// TIA Portal project "Szablon_Finał_V17" (V17)

(* hardware
DEVICE "S7-1200 station_1"  S7-1200 Station
   slot 0: "Rack_0"  S7-1200 Rack  Rack  V1.0
   slot 1: "PLC_1"  CPU 1214C DC/DC/DC  6ES7 214-1AG40-0XB0  V4.2
*)

// ===== PLC "PLC_1"  CPU 1214C DC/DC/DC =====

VAR_GLOBAL   // PLC tag table "Default tag table"
   "minimum" AT %I0.0 : Bool;
   "maksimum" AT %I0.1 : Bool;
   "poziom A" AT %I0.2 : Bool;
   "minimum B" AT %I0.3 : Bool;
   "Pokrywa" AT %I0.4 : Bool;
   "Start" AT %I0.5 : Bool;
   "Stop awaryjny" AT %I0.6 : Bool;
   "Zwolnij alarm" AT %I0.7 : Bool;
   "Mieszadło M1" AT %Q0.0 : Bool;
   "Mieszadło M2" AT %Q0.1 : Bool;
   "Zawór Z1" AT %Q0.2 : Bool;
   "Zawór Z2" AT %Q0.3 : Bool;
   "Zawór Z3" AT %Q0.4 : Bool;
   "Pompa P" AT %Q0.5 : Bool;
   "Alarm" AT %Q0.6 : Bool;
   "Tag_1" AT %MW50 : Int;
END_VAR

DATA_BLOCK "Dwa zbiorniki_DB"   // DB6
{ S7_Optimized_Access := 'TRUE' }
VERSION : 0.1
// stored: InstanceOfName Dwa zbiorniki
"Dwa zbiorniki"
BEGIN
END_DATA_BLOCK

DATA_BLOCK "Mieszanie substancji_DB"   // DB10
{ S7_Optimized_Access := 'TRUE' }
VERSION : 0.1
// stored: InstanceOfName Mieszanie substancji
"Mieszanie substancji"
BEGIN
END_DATA_BLOCK

// folder: System blocks/Program resources

DATA_BLOCK "IEC_Timer_0_DB"   // DB1
{ S7_Optimized_Access := 'TRUE' }
AUTHOR : Simatic
FAMILY : IEC
NAME : IEC_TMR
VERSION : 1.0
// stored: InstanceOfName IEC_TIMER
"IEC_TIMER"
BEGIN
END_DATA_BLOCK

DATA_BLOCK "IEC_Timer_0_DB_1"   // DB2
{ S7_Optimized_Access := 'TRUE' }
AUTHOR : Simatic
FAMILY : IEC
NAME : IEC_TMR
VERSION : 1.0
// stored: InstanceOfName IEC_TIMER
"IEC_TIMER"
BEGIN
END_DATA_BLOCK

DATA_BLOCK "IEC_Timer_0_DB_2"   // DB3
{ S7_Optimized_Access := 'TRUE' }
AUTHOR : Simatic
FAMILY : IEC
NAME : IEC_TMR
VERSION : 1.0
// stored: InstanceOfName IEC_TIMER
"IEC_TIMER"
BEGIN
END_DATA_BLOCK

DATA_BLOCK "IEC_Timer_0_DB_3"   // DB4
{ S7_Optimized_Access := 'TRUE' }
AUTHOR : Simatic
FAMILY : IEC
NAME : IEC_TMR
VERSION : 1.0
// stored: InstanceOfName IEC_TIMER
"IEC_TIMER"
BEGIN
END_DATA_BLOCK

DATA_BLOCK "IEC_Timer_0_DB_4"   // DB5
{ S7_Optimized_Access := 'TRUE' }
AUTHOR : Simatic
FAMILY : IEC
NAME : IEC_TMR
VERSION : 1.0
// stored: InstanceOfName IEC_TIMER
"IEC_TIMER"
BEGIN
END_DATA_BLOCK

DATA_BLOCK "IEC_Timer_0_DB_5"   // DB7
{ S7_Optimized_Access := 'TRUE' }
AUTHOR : Simatic
FAMILY : IEC
NAME : IEC_TMR
VERSION : 1.0
// stored: InstanceOfName IEC_TIMER
"IEC_TIMER"
BEGIN
END_DATA_BLOCK

DATA_BLOCK "IEC_Timer_0_DB_6"   // DB8
{ S7_Optimized_Access := 'TRUE' }
AUTHOR : Simatic
FAMILY : IEC
NAME : IEC_TMR
VERSION : 1.0
// stored: InstanceOfName IEC_TIMER
"IEC_TIMER"
BEGIN
END_DATA_BLOCK

DATA_BLOCK "IEC_Timer_0_DB_7"   // DB9
{ S7_Optimized_Access := 'TRUE' }
AUTHOR : Simatic
FAMILY : IEC
NAME : IEC_TMR
VERSION : 1.0
// stored: InstanceOfName IEC_TIMER
"IEC_TIMER"
BEGIN
END_DATA_BLOCK

// folder: (top level)

FUNCTION_BLOCK "Dwa zbiorniki"   // FB1, LAD
{ S7_Optimized_Access := 'TRUE' }
VERSION : 0.1
   VAR_INPUT
      minimum : Bool;
      maximum : Bool;
      "poziom A" : Bool;
      "minimum B" : Bool;
      Pokrywa : Bool;
      Start : Bool;
      "Stop awaryjny" : Bool;
      "Zwolnij alarm" : Bool;
   END_VAR
   VAR_OUTPUT
      M1 : Bool;
      M2 : Bool;
      "Pompa P" : Bool;
      Alarm : Bool;
   END_VAR
   VAR_IN_OUT
      Z1 : Bool;
      Z2 : Bool;
      Z3 : Bool;
      State : Int;
   END_VAR
   VAR
      Start_edge : Bool;
      Stop_awaryjny_edge : Bool;
      Zwolnij_alarm_edge : Bool;
   END_VAR
   VAR_TEMP
      "alarm 0_5Hz" : Bool;
      "alarm 1Hz" : Bool;
      alarm_awaryjny : Bool;
   END_VAR
   VAR_TEMP   // added for the SCL form of the ladder/FBD networks
      _w1 : Bool;
      _w2 : Bool;
   END_VAR
BEGIN

REGION Network 1
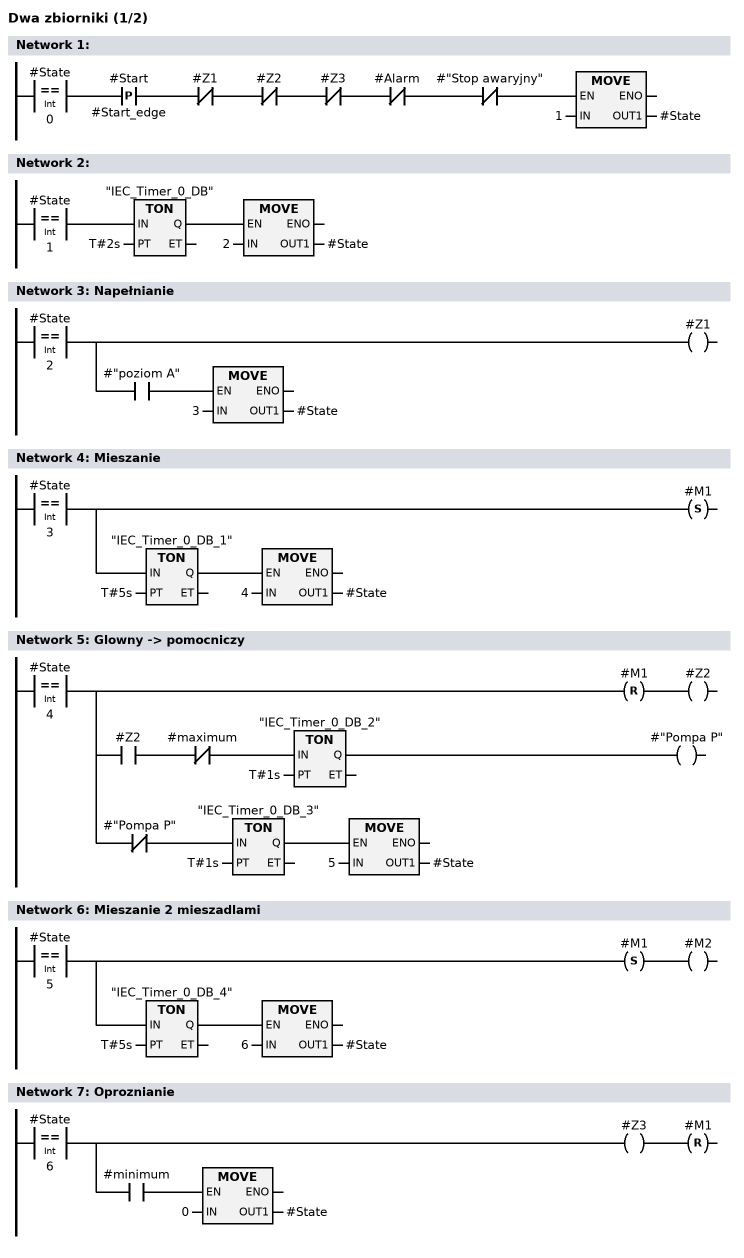
   RUNG wire#powerrail
      { S7_Templates := "SrcType := Int" } EQ_Contact(in1 := #State, in2 := 0)
      P_Contact(operand := #Start, bit := #Start_edge)
      I_Contact( #Z1 )
      I_Contact( #Z2 )
      I_Contact( #Z3 )
      I_Contact( #Alarm )
      I_Contact( #"Stop awaryjny" )
      Move(in := 1, out1 => #State)
   END_RUNG
   // the same network as SCL:
   #_w1 := (#State = 0) AND #Start AND NOT #Start_edge;   // rising edge of #Start
   #Start_edge := #Start;
   IF #_w1 AND NOT #Z1 AND NOT #Z2 AND NOT #Z3 AND NOT #Alarm AND NOT #"Stop awaryjny" THEN
       #State := 1;
   END_IF;
END_REGION

REGION Network 2
   "IEC_Timer_0_DB".TON(IN := #State = 1, PT := T#2s);
   IF "IEC_Timer_0_DB".Q THEN #State := 2; END_IF;
END_REGION

REGION Network 3: Napełnianie
   RUNG wire#powerrail
      { S7_Templates := "SrcType := Int" } EQ_Contact(in1 := #State, in2 := 2)
      wire#w1
      Coil( #Z1 )
   END_RUNG
   RUNG wire#w1
      Contact( #"poziom A" )
      Move(in := 3, out1 => #State)
   END_RUNG
   // the same network as SCL:
   #Z1 := #State = 2;
   IF #Z1 AND #"poziom A" THEN #State := 3; END_IF;
END_REGION

REGION Network 4: Mieszanie
   #_w1 := #State = 3;
   IF #_w1 THEN #M1 := TRUE; END_IF;
   "IEC_Timer_0_DB_1".TON(IN := #_w1, PT := T#5s);
   IF "IEC_Timer_0_DB_1".Q THEN #State := 4; END_IF;
END_REGION

REGION Network 5: Glowny -> pomocniczy
   #_w1 := #State = 4;
   IF #_w1 THEN #M1 := FALSE; END_IF;
   #Z2 := #_w1;
   "IEC_Timer_0_DB_2".TON(IN := #_w1 AND #Z2 AND NOT #maximum, PT := T#1s);
   #"Pompa P" := "IEC_Timer_0_DB_2".Q;
   "IEC_Timer_0_DB_3".TON(IN := #_w1 AND NOT #"Pompa P", PT := T#1s);
   IF "IEC_Timer_0_DB_3".Q THEN #State := 5; END_IF;
END_REGION

REGION Network 6: Mieszanie 2 mieszadlami
   #_w1 := #State = 5;
   IF #_w1 THEN #M1 := TRUE; END_IF;
   #M2 := #_w1;
   "IEC_Timer_0_DB_4".TON(IN := #_w1, PT := T#5s);
   IF "IEC_Timer_0_DB_4".Q THEN #State := 6; END_IF;
END_REGION

REGION Network 7: Oproznianie
   RUNG wire#powerrail
      { S7_Templates := "SrcType := Int" } EQ_Contact(in1 := #State, in2 := 6)
      wire#w1
      Coil( #Z3 )
      R_Coil( #M1 )
   END_RUNG
   RUNG wire#w1
      Contact( #minimum )
      Move(in := 0, out1 => #State)
   END_RUNG
   // the same network as SCL:
   #Z3 := #State = 6;
   IF #Z3 THEN #M1 := FALSE; END_IF;
   IF #Z3 AND #minimum THEN #State := 0; END_IF;
END_REGION

REGION Network 8: f = 0.5Hz, duty = 25%
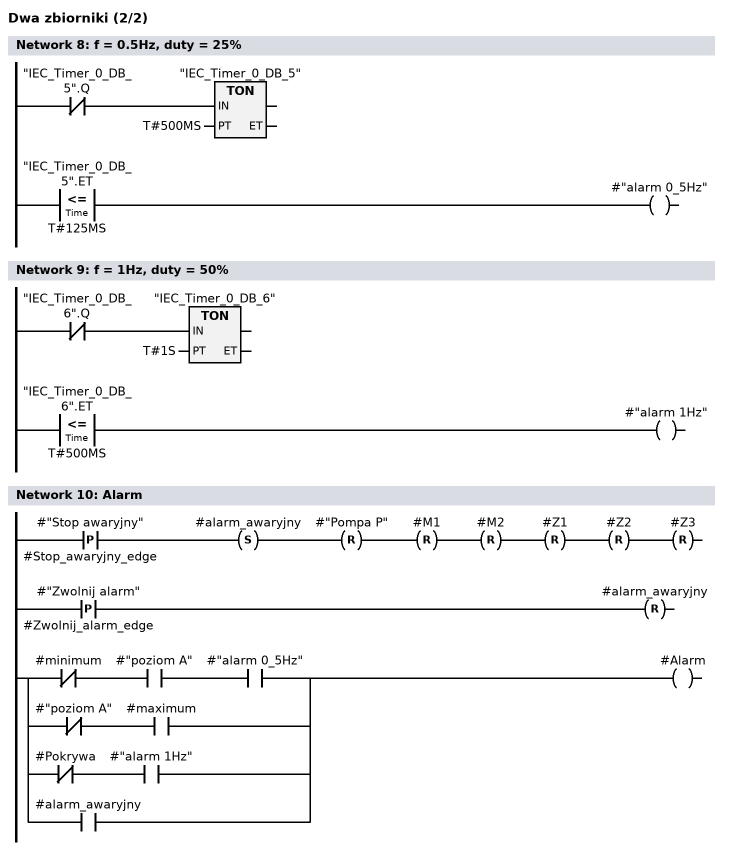
   "IEC_Timer_0_DB_5".TON(IN := NOT "IEC_Timer_0_DB_5".Q, PT := T#500MS);
   #"alarm 0_5Hz" := "IEC_Timer_0_DB_5".ET <= T#125MS;
END_REGION

REGION Network 9: f = 1Hz, duty = 50%
   "IEC_Timer_0_DB_6".TON(IN := NOT "IEC_Timer_0_DB_6".Q, PT := T#1S);
   #"alarm 1Hz" := "IEC_Timer_0_DB_6".ET <= T#500MS;
END_REGION

REGION Network 10: Alarm
   RUNG wire#powerrail
      P_Contact(operand := #"Stop awaryjny", bit := #Stop_awaryjny_edge)
      S_Coil( #alarm_awaryjny )
      R_Coil( #"Pompa P" )
      R_Coil( #M1 )
      R_Coil( #M2 )
      R_Coil( #Z1 )
      R_Coil( #Z2 )
      R_Coil( #Z3 )
   END_RUNG
   RUNG wire#powerrail
      P_Contact(operand := #"Zwolnij alarm", bit := #Zwolnij_alarm_edge)
      R_Coil( #alarm_awaryjny )
   END_RUNG
   RUNG wire#powerrail
      I_Contact( #minimum )
      Contact( #"poziom A" )
      Contact( #"alarm 0_5Hz" )
      wire#w1
      Coil( #Alarm )
   END_RUNG
   RUNG wire#powerrail
      I_Contact( #"poziom A" )
      Contact( #maximum )
   END_RUNG wire#w1
   RUNG wire#powerrail
      I_Contact( #Pokrywa )
      Contact( #"alarm 1Hz" )
   END_RUNG wire#w1
   RUNG wire#powerrail
      Contact( #alarm_awaryjny )
   END_RUNG wire#w1
   // the same network as SCL:
   #_w1 := #"Stop awaryjny" AND NOT #Stop_awaryjny_edge;   // rising edge of #"Stop awaryjny"
   #Stop_awaryjny_edge := #"Stop awaryjny";
   IF #_w1 THEN
       #alarm_awaryjny := TRUE;
       #"Pompa P" := FALSE;
       #M1 := FALSE;
       #M2 := FALSE;
       #Z1 := FALSE;
       #Z2 := FALSE;
       #Z3 := FALSE;
   END_IF;
   #_w2 := #"Zwolnij alarm" AND NOT #Zwolnij_alarm_edge;   // rising edge of #"Zwolnij alarm"
   #Zwolnij_alarm_edge := #"Zwolnij alarm";
   IF #_w2 THEN #alarm_awaryjny := FALSE; END_IF;
   #Alarm := (NOT #minimum AND #"poziom A" AND #"alarm 0_5Hz") OR (NOT #"poziom A" AND #maximum) OR (NOT #Pokrywa AND #"alarm 1Hz") OR #alarm_awaryjny;
END_REGION
END_FUNCTION_BLOCK

FUNCTION_BLOCK "Mieszanie substancji"   // FB2, LAD
{ S7_Optimized_Access := 'TRUE' }
VERSION : 0.1
   VAR_OUTPUT
      A_percent : Real;
      B_percent : Real;
      C_percent : Real;
      AF001 : Bool;
      AF002 : Bool;
      AF003 : Bool;
      AF004 : Bool;
      AF005 : Bool;
      AF006 : Bool;
      AF007 : Bool;
      AF008 : Bool;
   END_VAR
   VAR_IN_OUT
      A_value : Int := 2500;
      B_value : Int := 2500;
      C_value : Int := 9000;
      M_value : Int := 12;
   END_VAR
   VAR
      TON_Out : Bool;
      State : Int;
      TON_Out_edge : Bool;
      A_in_M : Int;
      B_in_M : Int;
      C_in_M : Int;
      TON_Out_edge2 : Bool;
   END_VAR
   VAR CONSTANT
      qa : Int := 4;
      qb : Int := 8;
      qc : Int := 12;
      qabc : Int := 15;
   END_VAR
   VAR_TEMP   // added for the SCL form of the ladder/FBD networks
      _w1 : Bool;
      _w2 : Bool;
   END_VAR
BEGIN

REGION Network 1
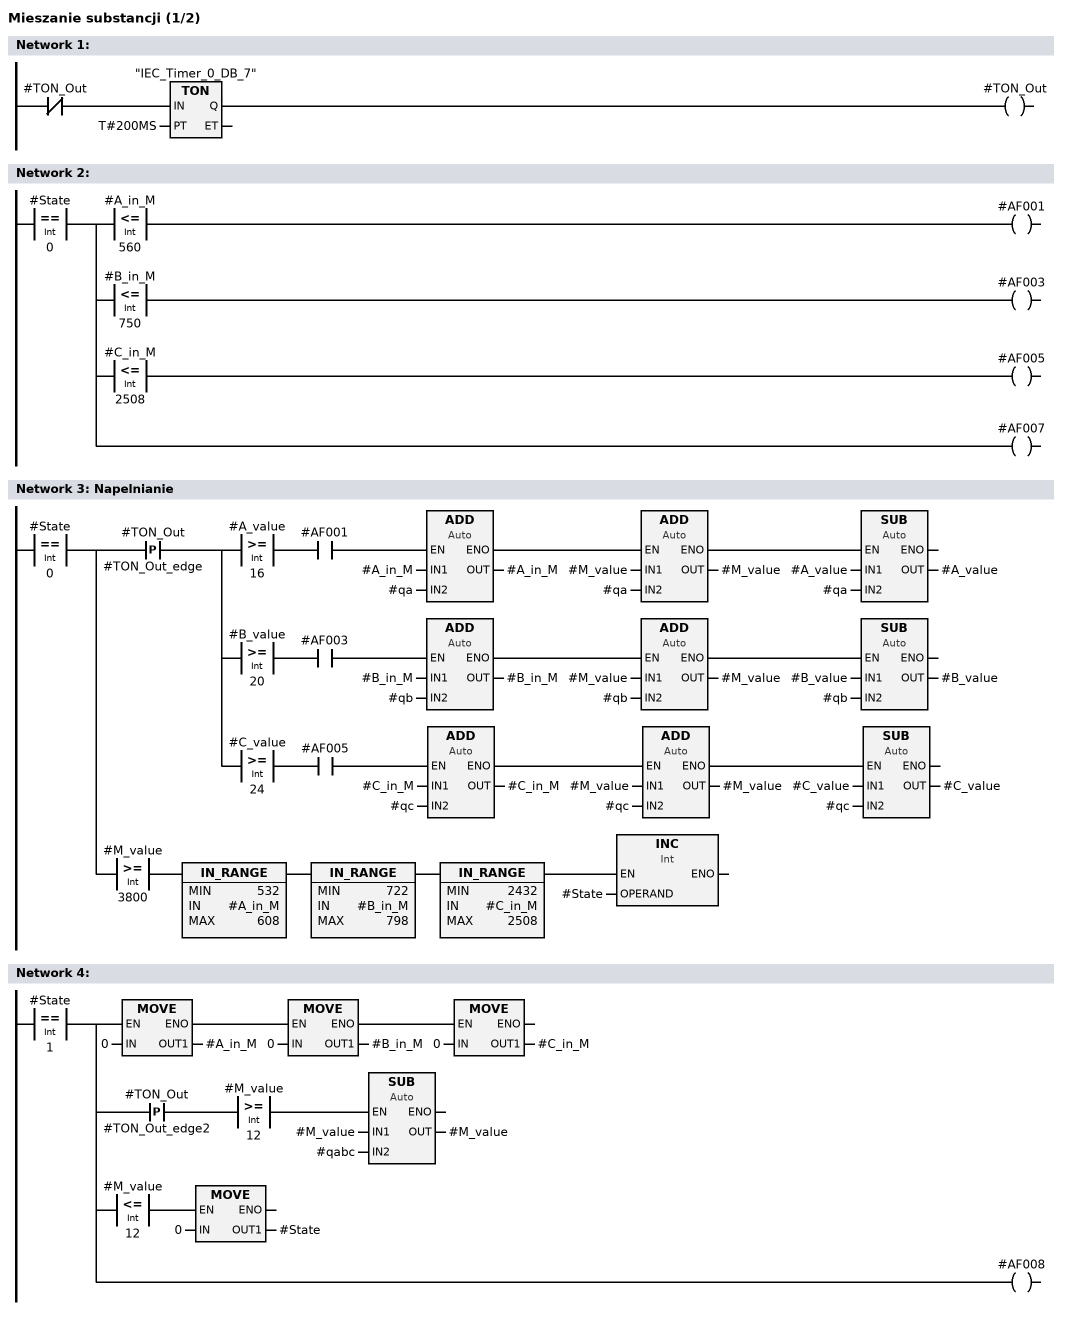
   "IEC_Timer_0_DB_7".TON(IN := NOT #TON_Out, PT := T#200MS);
   #TON_Out := "IEC_Timer_0_DB_7".Q;
END_REGION

REGION Network 2
   RUNG wire#powerrail
      { S7_Templates := "SrcType := Int" } EQ_Contact(in1 := #State, in2 := 0)
      wire#w1
      { S7_Templates := "SrcType := Int" } LE_Contact(in1 := #A_in_M, in2 := 560)
      Coil( #AF001 )
   END_RUNG
   RUNG wire#w1
      { S7_Templates := "SrcType := Int" } LE_Contact(in1 := #B_in_M, in2 := 750)
      Coil( #AF003 )
   END_RUNG
   RUNG wire#w1
      { S7_Templates := "SrcType := Int" } LE_Contact(in1 := #C_in_M, in2 := 2508)
      Coil( #AF005 )
   END_RUNG
   RUNG wire#w1
      Coil( #AF007 )
   END_RUNG
   // the same network as SCL:
   #_w1 := #State = 0;
   #AF001 := #_w1 AND (#A_in_M <= 560);
   #AF003 := #_w1 AND (#B_in_M <= 750);
   #AF005 := #_w1 AND (#C_in_M <= 2508);
   #AF007 := #_w1;
END_REGION

REGION Network 3: Napelnianie
   RUNG wire#powerrail
      { S7_Templates := "SrcType := Int" } EQ_Contact(in1 := #State, in2 := 0)
      wire#w1
      P_Contact(operand := #TON_Out, bit := #TON_Out_edge)
      wire#w2
      { S7_Templates := "SrcType := Int" } GE_Contact(in1 := #A_value, in2 := 16)
      Contact( #AF001 )
      Add(in1 := #A_in_M, in2 := #qa, out => #A_in_M)
      Add(in1 := #M_value, in2 := #qa, out => #M_value)
      Sub(in1 := #A_value, in2 := #qa, out => #A_value)
   END_RUNG
   RUNG wire#w2
      { S7_Templates := "SrcType := Int" } GE_Contact(in1 := #B_value, in2 := 20)
      Contact( #AF003 )
      Add(in1 := #B_in_M, in2 := #qb, out => #B_in_M)
      Add(in1 := #M_value, in2 := #qb, out => #M_value)
      Sub(in1 := #B_value, in2 := #qb, out => #B_value)
   END_RUNG
   RUNG wire#w2
      { S7_Templates := "SrcType := Int" } GE_Contact(in1 := #C_value, in2 := 24)
      Contact( #AF005 )
      Add(in1 := #C_in_M, in2 := #qc, out => #C_in_M)
      Add(in1 := #M_value, in2 := #qc, out => #M_value)
      Sub(in1 := #C_value, in2 := #qc, out => #C_value)
   END_RUNG
   RUNG wire#w1
      { S7_Templates := "SrcType := Int" } GE_Contact(in1 := #M_value, in2 := 3800)
      { S7_Templates := "SrcType := Int" } InRange(min := 532, in := #A_in_M, max := 608)
      { S7_Templates := "SrcType := Int" } InRange(min := 722, in := #B_in_M, max := 798)
      { S7_Templates := "SrcType := Int" } InRange(min := 2432, in := #C_in_M, max := 2508)
      { S7_Templates := "DestType := Int" } Inc( #State )
   END_RUNG
   // the same network as SCL:
   #_w1 := #State = 0;
   #_w2 := #_w1 AND #TON_Out AND NOT #TON_Out_edge;   // rising edge of #TON_Out
   #TON_Out_edge := #TON_Out;
   IF #_w2 AND (#A_value >= 16) AND #AF001 THEN
       #A_in_M := #A_in_M + #qa;
       #M_value := #M_value + #qa;
       #A_value := #A_value - #qa;
   END_IF;
   IF #_w2 AND (#B_value >= 20) AND #AF003 THEN
       #B_in_M := #B_in_M + #qb;
       #M_value := #M_value + #qb;
       #B_value := #B_value - #qb;
   END_IF;
   IF #_w2 AND (#C_value >= 24) AND #AF005 THEN
       #C_in_M := #C_in_M + #qc;
       #M_value := #M_value + #qc;
       #C_value := #C_value - #qc;
   END_IF;
   IF #_w1 AND (#M_value >= 3800) AND (532 <= #A_in_M) AND (#A_in_M <= 608) AND (722 <= #B_in_M) AND (#B_in_M <= 798) AND (2432 <= #C_in_M) AND (#C_in_M <= 2508) THEN
       #State := #State + 1;
   END_IF;
END_REGION

REGION Network 4
   RUNG wire#powerrail
      { S7_Templates := "SrcType := Int" } EQ_Contact(in1 := #State, in2 := 1)
      wire#w1
      Move(in := 0, out1 => #A_in_M)
      Move(in := 0, out1 => #B_in_M)
      Move(in := 0, out1 => #C_in_M)
   END_RUNG
   RUNG wire#w1
      P_Contact(operand := #TON_Out, bit := #TON_Out_edge2)
      { S7_Templates := "SrcType := Int" } GE_Contact(in1 := #M_value, in2 := 12)
      Sub(in1 := #M_value, in2 := #qabc, out => #M_value)
   END_RUNG
   RUNG wire#w1
      { S7_Templates := "SrcType := Int" } LE_Contact(in1 := #M_value, in2 := 12)
      Move(in := 0, out1 => #State)
   END_RUNG
   RUNG wire#w1
      Coil( #AF008 )
   END_RUNG
   // the same network as SCL:
   #_w1 := #State = 1;
   IF #_w1 THEN
       #A_in_M := 0;
       #B_in_M := 0;
       #C_in_M := 0;
   END_IF;
   #_w2 := #_w1 AND #TON_Out AND NOT #TON_Out_edge2;   // rising edge of #TON_Out
   #TON_Out_edge2 := #TON_Out;
   IF #_w2 AND (#M_value >= 12) THEN #M_value := #M_value - #qabc; END_IF;
   IF #_w1 AND (#M_value <= 12) THEN #State := 0; END_IF;
   #AF008 := #_w1;
END_REGION

REGION Network 5
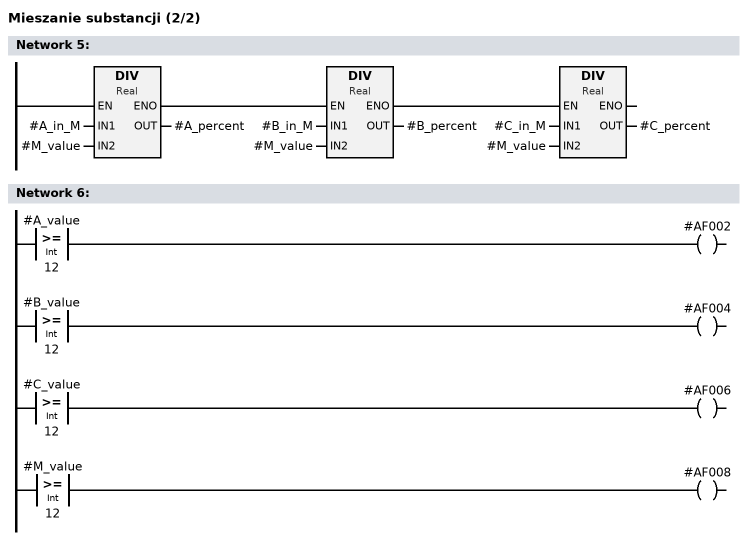
   RUNG wire#powerrail
      { S7_Templates := "SrcType := Real" } Div(in1 := #A_in_M, in2 := #M_value, out => #A_percent)
      { S7_Templates := "SrcType := Real" } Div(in1 := #B_in_M, in2 := #M_value, out => #B_percent)
      { S7_Templates := "SrcType := Real" } Div(in1 := #C_in_M, in2 := #M_value, out => #C_percent)
   END_RUNG
   // the same network as SCL:
   #A_percent := #A_in_M / #M_value;
   #B_percent := #B_in_M / #M_value;
   #C_percent := #C_in_M / #M_value;
END_REGION

REGION Network 6
   RUNG wire#powerrail
      { S7_Templates := "SrcType := Int" } GE_Contact(in1 := #A_value, in2 := 12)
      Coil( #AF002 )
   END_RUNG
   RUNG wire#powerrail
      { S7_Templates := "SrcType := Int" } GE_Contact(in1 := #B_value, in2 := 12)
      Coil( #AF004 )
   END_RUNG
   RUNG wire#powerrail
      { S7_Templates := "SrcType := Int" } GE_Contact(in1 := #C_value, in2 := 12)
      Coil( #AF006 )
   END_RUNG
   RUNG wire#powerrail
      { S7_Templates := "SrcType := Int" } GE_Contact(in1 := #M_value, in2 := 12)
      Coil( #AF008 )
   END_RUNG
   // the same network as SCL:
   #AF002 := #A_value >= 12;
   #AF004 := #B_value >= 12;
   #AF006 := #C_value >= 12;
   #AF008 := #M_value >= 12;
END_REGION
END_FUNCTION_BLOCK

ORGANIZATION_BLOCK "Main"   // OB1, LAD, ProgramCycle
TITLE = "Main Program Sweep (Cycle)"
{ S7_Optimized_Access := 'TRUE' }
VERSION : 0.1
   VAR_INPUT
      Initial_Call : Bool;   // Initial call of this OB
      Remanence : Bool;   // =True, if remanent data are available
   END_VAR
BEGIN

REGION Network 1
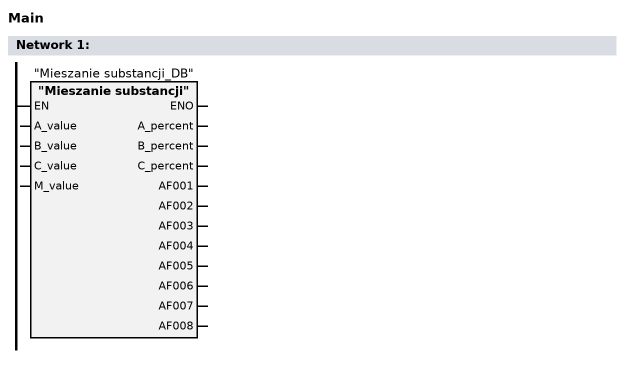
   RUNG wire#powerrail
      "Mieszanie substancji_DB"(A_value :=, B_value :=, C_value :=, M_value :=, A_percent =>, B_percent =>, C_percent =>, AF001 =>, AF002 =>, AF003 =>, AF004 =>, AF005 =>, AF006 =>, AF007 =>, AF008 =>)
   END_RUNG
   // the same network as SCL:
   "Mieszanie substancji_DB"();   // "Mieszanie substancji"
END_REGION
END_ORGANIZATION_BLOCK